FUNCTION_BLOCK Printr
  (* Standard: 61499-2 *)
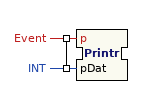
  EVENT_INPUT
    p WITH pDat;
  END_EVENT
  VAR_INPUT
    pDat : INT;
  END_VAR
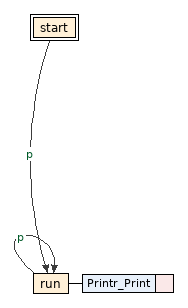
  EC_STATES
    start;
    run : Printr_Print;
  END_STATES
  EC_TRANSITIONS
    start TO run := p;
    run TO run := p;
  END_TRANSITIONS
  ALGORITHM Printr_Print IN C:
printf("val: %i\n", me->pDat);
  END_ALGORITHM
END_FUNCTION_BLOCK
